// TIA Portal project "pinmachine_vimpr" (V16)

(* hardware
DEVICE "S7-1200 station_1"  S7-1200 Station
   slot 0: "Rack_0"  S7-1200 Rack  Rack  V1.0
   slot 1: "PLC_1"  CPU 1212C DC/DC/DC  6ES7 212-1AE40-0XB0  V4.4
   slot 2: "DI 16x24VDC_1"  6ES7 221-1BH32-0XB0  V2.0
*)

// ===== PLC "PLC_1"  CPU 1212C DC/DC/DC =====

VAR_GLOBAL   // PLC tag table "Default tag table"
   "Cyc1_Top1_Act" AT %I0.0 : Bool;
   "Cyc2_Top1_Act" AT %I0.1 : Bool;
   "Cyc3_Top1_Act" AT %I0.2 : Bool;
   "Cyc4_Top1_Act" AT %I0.3 : Bool;
   "Cyc1_Bot1_Act" AT %I0.4 : Bool;
   "Cyc2_Bot1_Act" AT %I0.5 : Bool;
   "Cyc3_Bot1_Act" AT %I0.6 : Bool;
   "Cyc4_Bot1_Act" AT %I0.7 : Bool;
   "CycHold_Rep" AT %I1.0 : Bool;
   "CycHold_Act" AT %I1.1 : Bool;
   "Cyc1_Top2_Act" AT %I1.2 : Bool;
   "Cyc2_Top2_Act" AT %I1.3 : Bool;
   "Cyc3_Top2_Act" AT %I1.4 : Bool;
   "Cyc4_Top2_Act" AT %I1.5 : Bool;
   "Cyc5_Top2_Act" AT %I1.6 : Bool;
   "Cyc1_Bot2_Act" AT %I1.7 : Bool;
   "Cyc2_Bot2_Act" AT %I2.0 : Bool;
   "Cyc3_Bot2_Act" AT %I2.1 : Bool;
   "Cyc4_Bot2_Act" AT %I2.2 : Bool;
   "Cyc5_Bot2_Act" AT %I2.3 : Bool;
   "Foot_Switch" AT %I2.4 : Bool;
   "4_Part_Detect" AT %I2.5 : Bool;
   "5_Part_Detect" AT %I2.6 : Bool;
   "Safety_Sensor" AT %I2.7 : Bool;
   "QValve4" AT %Q0.0 : Bool;
   "QValve5" AT %Q0.1 : Bool;
   "QHold4" AT %Q0.2 : Bool;
   "QHold5" AT %Q0.3 : Bool;
   "QValveHolder" AT %Q0.4 : Bool;
   "QValveBuzzer" AT %Q0.5 : Bool;
   "MValve4" AT %M0.0 : Bool;
   "MValve5" AT %M0.1 : Bool;
   "MHold4" AT %M0.2 : Bool;
   "MHold5" AT %M0.3 : Bool;
   "x" AT %M0.4 : Bool;
   "MBuzzer" AT %M0.5 : Bool;
   "MBussy" AT %M0.6 : Bool;
   "MDone" AT %M0.7 : Bool;
   "Start" AT %M1.0 : Bool;
   "Auto" AT %M1.1 : Bool;
   "Run" AT %M1.2 : Bool;
   "Timer_Alarm" AT %MD0 : Time;
   "Timer_4Cyl" AT %MD20 : Time;
   "Timer_5Cyl" AT %MD21 : Time;
   "DoneCheckSSBot1" AT %M9.0 : Bool;
   "DoneCheckSSTop1" AT %M9.1 : Bool;
   "DoneCheckSSBot2" AT %M9.2 : Bool;
   "DoneCheckSSTop2" AT %M9.3 : Bool;
   "Alarm" AT %M9.4 : Bool;
   "Cyc1_Top1_Act_Alarm" AT %M9.5 : Bool;
   "Cyc2_Top1_Act_Alarm" AT %M9.6 : Bool;
   "Cyc3_Top1_Act_Alarm" AT %M9.7 : Bool;
   "Cyc4_Top1_Act_Alarm" AT %M10.0 : Bool;
   "Cyc1_Bot1_Act_Alarm" AT %M10.1 : Bool;
   "Cyc2_Bot1_Act_Alarm" AT %M10.2 : Bool;
   "Cyc3_Bot1_Act_Alarm" AT %M10.3 : Bool;
   "Cyc4_Bot1_Act_Alarm" AT %M10.4 : Bool;
   "Cyc1_Bot2_Act_Alarm" AT %M10.5 : Bool;
   "Cyc2_Bot2_Act_Alarm" AT %M10.6 : Bool;
   "Cyc3_Bot2_Act_Alarm" AT %M10.7 : Bool;
   "Cyc4_Bot2_Act_Alarm" AT %M11.0 : Bool;
   "Cyc5_Bot2_Act_Alarm" AT %M11.1 : Bool;
   "Cyc1_Top2_Act_Alarm" AT %M11.2 : Bool;
   "Cyc2_Top2_Act_Alarm" AT %M11.3 : Bool;
   "Cyc3_Top2_Act_Alarm" AT %M11.4 : Bool;
   "Cyc4_Top2_Act_Alarm" AT %M11.5 : Bool;
   "Cyc5_Top2_Act_Alarm" AT %M11.6 : Bool;
   "ResetAlarm" AT %M11.7 : Bool;
   "Step" AT %MW12 : Int;
   "4_Done" AT %M14.0 : Bool;
   "5_Done" AT %M14.1 : Bool;
   "Tag_1" AT %M1000.0 : Bool;
   "Tag_2" AT %M1000.1 : Bool;
   "Tag_3" AT %M1000.3 : Bool;
   "Tag_4" AT %M14.2 : Bool;
   "Tag_5" AT %M14.3 : Bool;
   "Count" AT %MW16 : Int;
   "Tag_6" AT %M1000.4 : Bool;
   "Tag_7" AT %M1000.5 : Bool;
   "Tag_8" AT %M1000.6 : Bool;
   "Tag_9" AT %M1000.7 : Bool;
   "Tag_10" AT %M1001.0 : Bool;
   "Tag_11" AT %M1001.2 : Bool;
   "Tag_12" AT %M1005.1 : Bool;
   "Tag_13" AT %M1005.2 : Bool;
   "Tag_14" AT %M1001.7 : Bool;
   "Tag_15" AT %M1001.6 : Bool;
   "Tag_16" AT %M1007.0 : Bool;
   "Tag_17" AT %M1007.1 : Bool;
END_VAR

DATA_BLOCK "TimerDB"   // DB6
{ S7_Optimized_Access := 'TRUE' }
VERSION : 0.1
   VAR RETAIN
      TimerCyl4_1 : DInt := 1000;
      TimerCyl4_2 : DInt := 1000;
      TimerCyl4_3 : DInt := 1000;
      TimerCyl4_4 : DInt := 1000;
      TimerCyl5_1 : DInt := 1000;
      TimerCyl5_2 : DInt := 1000;
      TimerCyl5_3 : DInt := 1000;
      TimerCyl5_4 : DInt := 1000;
      Timer_Safety : DInt := 5000;
   END_VAR
BEGIN
END_DATA_BLOCK

DATA_BLOCK "AlarmDB"   // DB7
{ S7_Optimized_Access := 'TRUE' }
VERSION : 0.1
   VAR
      Cyc1_Bot1_Act_Alarm : Bool;
      Cyc1_Bot2_Act_Alarm : Bool;
      Cyc1_Bot3_Act_Alarm : Bool;
      Cyc1_Bot4_Act_Alarm : Bool;
      Cyc1_Top1_Act_Alarm : Bool;
      Cyc1_Top2_Act_Alarm : Bool;
      Cyc1_Top3_Act_Alarm : Bool;
      Cyc1_Top4_Act_Alarm : Bool;
      Cyc2_Bot1_Act_Alarm : Bool;
      Cyc2_Bot2_Act_Alarm : Bool;
      Cyc2_Bot3_Act_Alarm : Bool;
      Cyc2_Bot4_Act_Alarm : Bool;
      Cyc2_Bot5_Act_Alarm : Bool;
      Cyc2_Top1_Act_Alarm : Bool;
      Cyc2_Top2_Act_Alarm : Bool;
      Cyc2_Top3_Act_Alarm : Bool;
      Cyc2_Top4_Act_Alarm : Bool;
      Cyc2_Top5_Act_Alarm : Bool;
      Sensor_Detect_4 : Bool;
      Sensor_Detect_5 : Bool;
      Sensor_Safety : Bool;
   END_VAR
BEGIN
END_DATA_BLOCK

// folder: System blocks/Program resources

DATA_BLOCK "TimerDone45"   // DB1
{ S7_Optimized_Access := 'TRUE' }
AUTHOR : Simatic
FAMILY : IEC
NAME : IEC_TMR
VERSION : 1.0
// stored: InstanceOfName IEC_TIMER
"IEC_TIMER"
BEGIN
END_DATA_BLOCK

DATA_BLOCK "TimerError"   // DB5
{ S7_Optimized_Access := 'TRUE' }
AUTHOR : Simatic
FAMILY : IEC
NAME : IEC_TMR
VERSION : 1.0
// stored: InstanceOfName IEC_TIMER
"IEC_TIMER"
BEGIN
END_DATA_BLOCK

DATA_BLOCK "TimerResetAlarm"   // DB16
{ S7_Optimized_Access := 'TRUE' }
AUTHOR : Simatic
FAMILY : IEC
NAME : IEC_TMR
VERSION : 1.0
// stored: InstanceOfName IEC_TIMER
"IEC_TIMER"
BEGIN
END_DATA_BLOCK

DATA_BLOCK "TimerResetStep"   // DB17
{ S7_Optimized_Access := 'TRUE' }
AUTHOR : Simatic
FAMILY : IEC
NAME : IEC_TMR
VERSION : 1.0
// stored: InstanceOfName IEC_TIMER
"IEC_TIMER"
BEGIN
END_DATA_BLOCK

// folder: (top level)

ORGANIZATION_BLOCK "Main"   // OB1, LAD, ProgramCycle
TITLE = "Main Program Sweep (Cycle)"
{ S7_Optimized_Access := 'TRUE' }
VERSION : 0.1
   VAR_INPUT
      Initial_Call : Bool;   // Initial call of this OB
      Remanence : Bool;   // =True, if remanent data are available
   END_VAR
   VAR_TEMP   // added for the SCL form of the ladder/FBD networks
      _w1 : Bool;
      _w2 : Bool;
      _w3 : Bool;
      _w4 : Bool;
      _w5 : Bool;
   END_VAR
BEGIN

REGION Network 1: Cycle
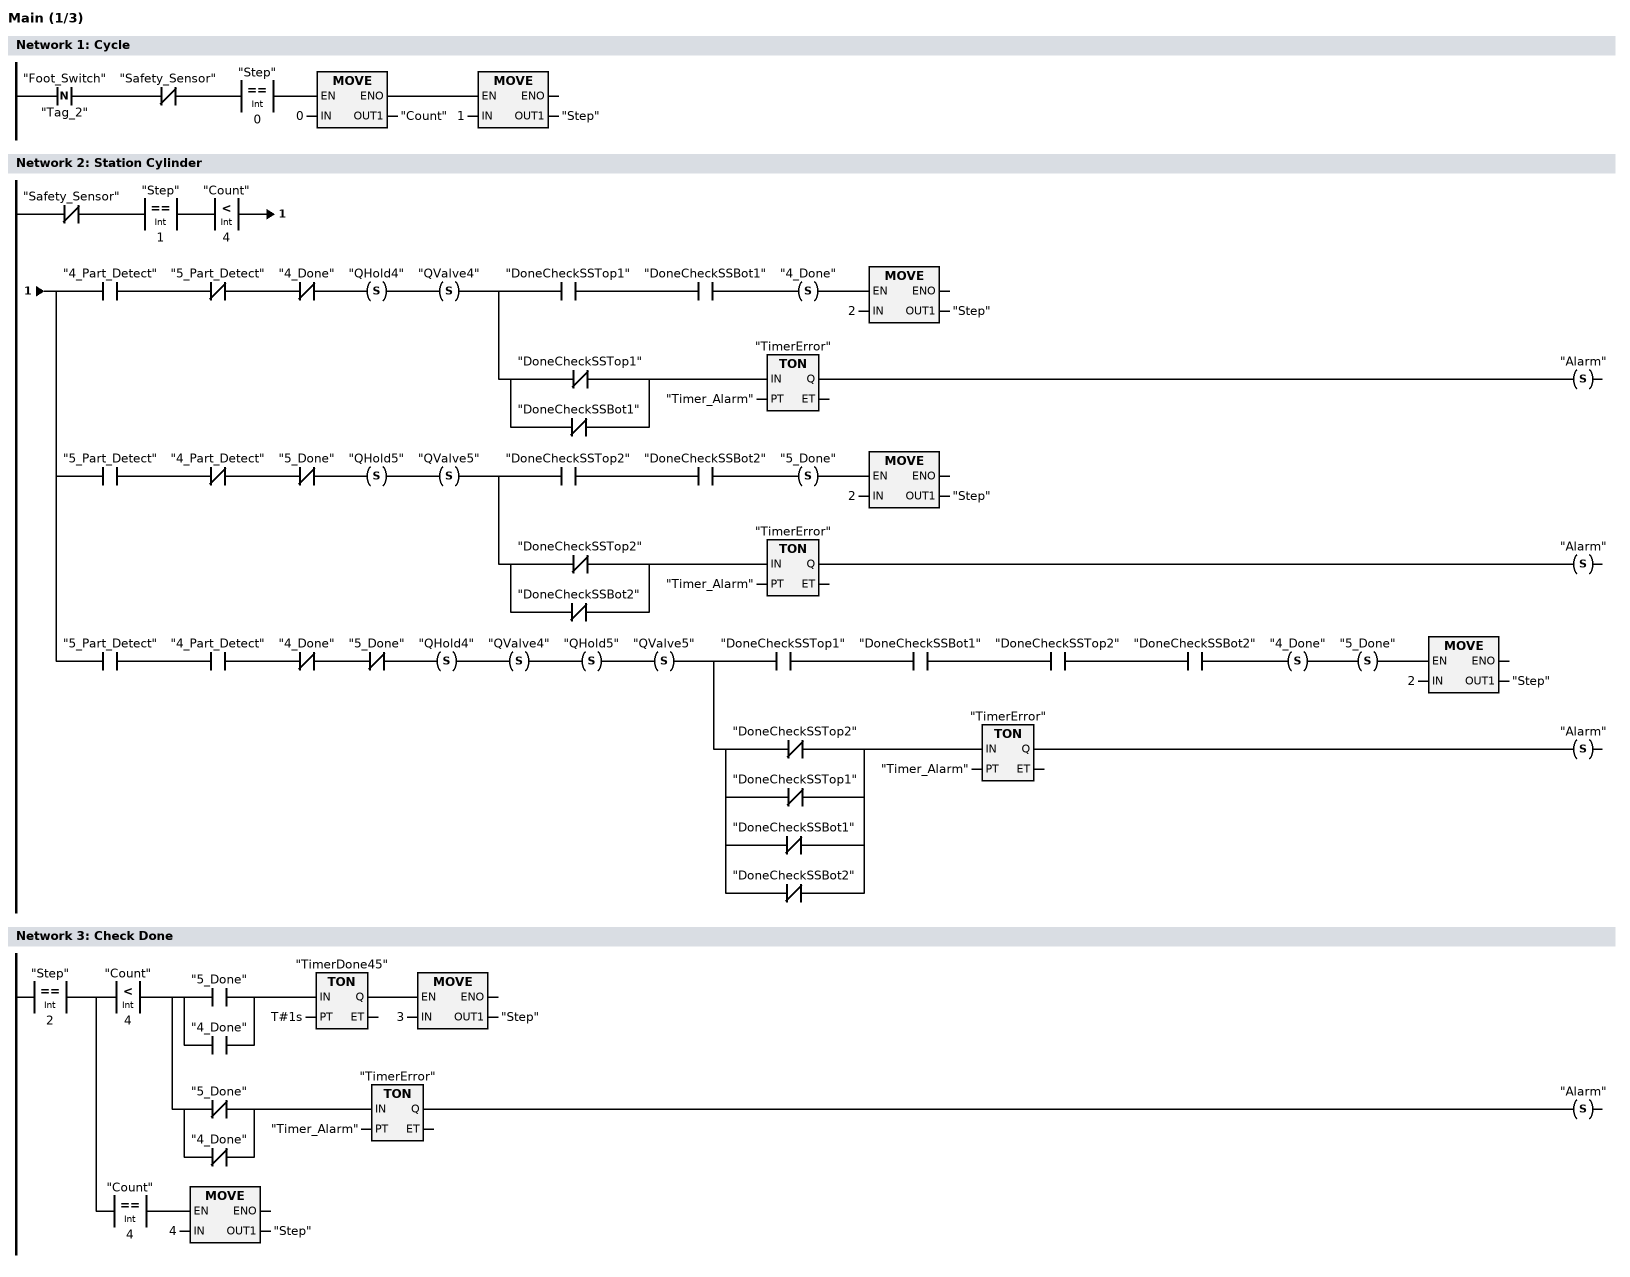
   RUNG wire#powerrail
      N_Contact(operand := "Foot_Switch", bit := "Tag_2")
      I_Contact( "Safety_Sensor" )
      { S7_Templates := "SrcType := Int" } EQ_Contact(in1 := "Step", in2 := 0)
      Move(in := 0, out1 => "Count")
      Move(in := 1, out1 => "Step")
   END_RUNG
   // the same network as SCL:
   #_w1 := NOT "Foot_Switch" AND "Tag_2";   // falling edge of "Foot_Switch"
   "Tag_2" := "Foot_Switch";
   IF #_w1 AND NOT "Safety_Sensor" AND ("Step" = 0) THEN
       "Count" := 0;
       "Step" := 1;
   END_IF;
END_REGION

REGION Network 2: Station Cylinder
   #_w1 := NOT "Safety_Sensor" AND ("Step" = 1) AND ("Count" < 4);
   #_w2 := #_w1 AND "4_Part_Detect" AND NOT "5_Part_Detect" AND NOT "4_Done";
   IF #_w2 THEN
       "QHold4" := TRUE;
       "QValve4" := TRUE;
   END_IF;
   IF #_w2 AND "DoneCheckSSTop1" AND "DoneCheckSSBot1" THEN
       "4_Done" := TRUE;
       "Step" := 2;
   END_IF;
   "TimerError".TON(IN := #_w2 AND (NOT "DoneCheckSSTop1" OR NOT "DoneCheckSSBot1"), PT := "Timer_Alarm");
   IF "TimerError".Q THEN "Alarm" := TRUE; END_IF;
   #_w3 := #_w1 AND "5_Part_Detect" AND NOT "4_Part_Detect" AND NOT "5_Done";
   IF #_w3 THEN
       "QHold5" := TRUE;
       "QValve5" := TRUE;
   END_IF;
   IF #_w3 AND "DoneCheckSSTop2" AND "DoneCheckSSBot2" THEN
       "5_Done" := TRUE;
       "Step" := 2;
   END_IF;
   "TimerError".TON(IN := #_w3 AND (NOT "DoneCheckSSTop2" OR NOT "DoneCheckSSBot2"), PT := "Timer_Alarm");
   IF "TimerError".Q THEN "Alarm" := TRUE; END_IF;
   #_w4 := #_w1 AND "5_Part_Detect" AND "4_Part_Detect" AND NOT "4_Done" AND NOT "5_Done";
   IF #_w4 THEN
       "QHold4" := TRUE;
       "QValve4" := TRUE;
       "QHold5" := TRUE;
       "QValve5" := TRUE;
   END_IF;
   IF #_w4 AND "DoneCheckSSTop1" AND "DoneCheckSSBot1" AND "DoneCheckSSTop2" AND "DoneCheckSSBot2" THEN
       "4_Done" := TRUE;
       "5_Done" := TRUE;
       "Step" := 2;
   END_IF;
   "TimerError".TON(IN := #_w4 AND (NOT "DoneCheckSSTop2" OR NOT "DoneCheckSSTop1" OR NOT "DoneCheckSSBot1" OR NOT "DoneCheckSSBot2"),
                    PT := "Timer_Alarm");
   IF "TimerError".Q THEN "Alarm" := TRUE; END_IF;
END_REGION

REGION Network 3: Check Done
   #_w1 := "Step" = 2;
   #_w2 := #_w1 AND ("Count" < 4);
   "TimerDone45".TON(IN := #_w2 AND ("5_Done" OR "4_Done"), PT := T#1s);
   IF "TimerDone45".Q THEN "Step" := 3; END_IF;
   "TimerError".TON(IN := #_w2 AND (NOT "5_Done" OR NOT "4_Done"), PT := "Timer_Alarm");
   IF "TimerError".Q THEN "Alarm" := TRUE; END_IF;
   IF #_w1 AND ("Count" = 4) THEN "Step" := 4; END_IF;
END_REGION

REGION Network 4: Step Reset Valve
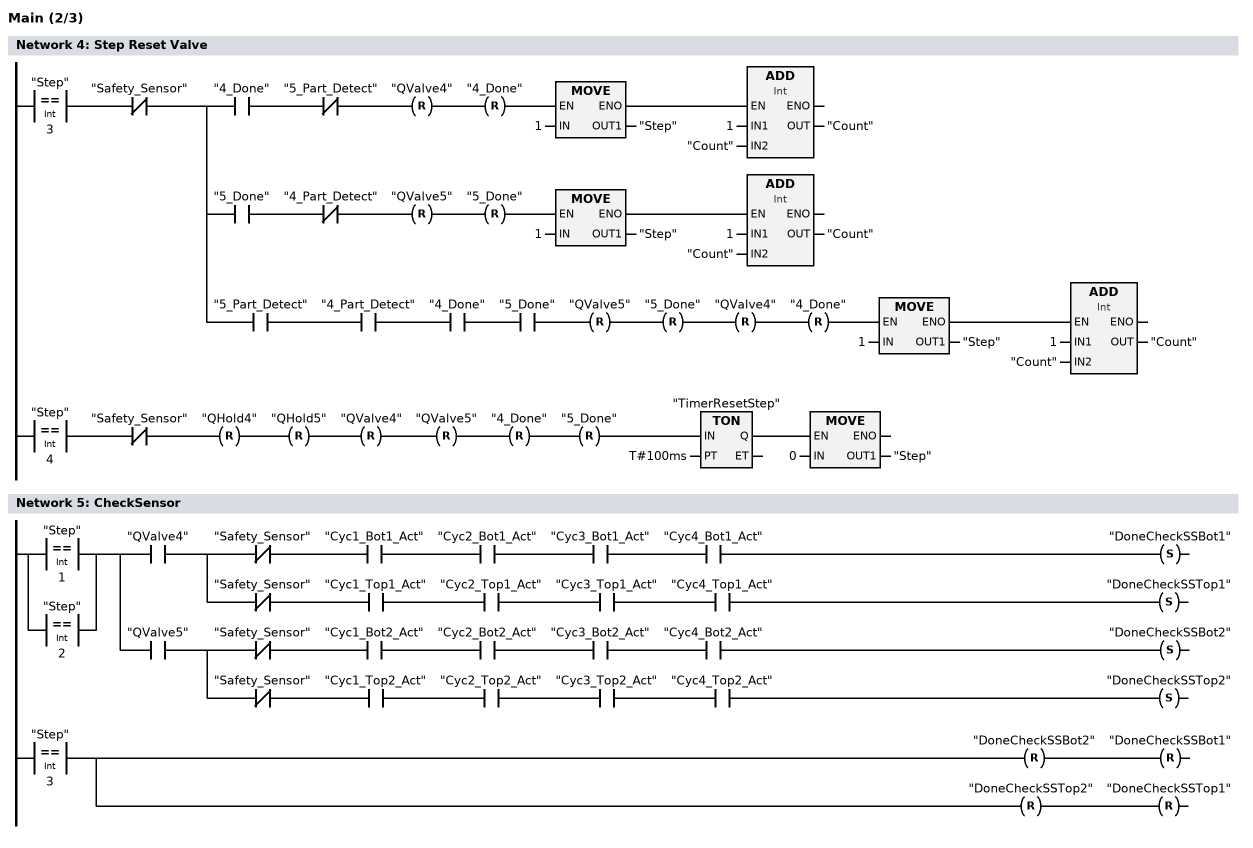
   #_w1 := ("Step" = 3) AND NOT "Safety_Sensor";
   IF #_w1 AND "4_Done" AND NOT "5_Part_Detect" THEN "QValve4" := FALSE; END_IF;
   #_w2 := #_w1 AND "4_Done" AND NOT "5_Part_Detect";
   IF #_w2 THEN
       "4_Done" := FALSE;
       "Step" := 1;
       "Count" := 1 + "Count";
   END_IF;
   IF #_w1 AND "5_Done" AND NOT "4_Part_Detect" THEN "QValve5" := FALSE; END_IF;
   #_w3 := #_w1 AND "5_Done" AND NOT "4_Part_Detect";
   IF #_w3 THEN
       "5_Done" := FALSE;
       "Step" := 1;
       "Count" := 1 + "Count";
   END_IF;
   IF #_w1 AND "5_Part_Detect" AND "4_Part_Detect" AND "4_Done" AND "5_Done" THEN "QValve5" := FALSE; END_IF;
   #_w4 := #_w1 AND "5_Part_Detect" AND "4_Part_Detect" AND "4_Done" AND "5_Done";
   IF #_w4 THEN
       "5_Done" := FALSE;
       "QValve4" := FALSE;
       "4_Done" := FALSE;
       "Step" := 1;
       "Count" := 1 + "Count";
   END_IF;
   #_w5 := ("Step" = 4) AND NOT "Safety_Sensor";
   IF #_w5 THEN
       "QHold4" := FALSE;
       "QHold5" := FALSE;
       "QValve4" := FALSE;
       "QValve5" := FALSE;
       "4_Done" := FALSE;
       "5_Done" := FALSE;
   END_IF;
   "TimerResetStep".TON(IN := #_w5, PT := T#100ms);
   IF "TimerResetStep".Q THEN "Step" := 0; END_IF;
END_REGION

REGION Network 5: CheckSensor
   RUNG wire#powerrail
      { S7_Templates := "SrcType := Int" } EQ_Contact(in1 := "Step", in2 := 1)
      wire#w1
      Contact( "QValve4" )
      wire#w2
      I_Contact( "Safety_Sensor" )
      Contact( "Cyc1_Bot1_Act" )
      Contact( "Cyc2_Bot1_Act" )
      Contact( "Cyc3_Bot1_Act" )
      Contact( "Cyc4_Bot1_Act" )
      S_Coil( "DoneCheckSSBot1" )
   END_RUNG
   RUNG wire#powerrail
      { S7_Templates := "SrcType := Int" } EQ_Contact(in1 := "Step", in2 := 2)
   END_RUNG wire#w1
   RUNG wire#w2
      I_Contact( "Safety_Sensor" )
      Contact( "Cyc1_Top1_Act" )
      Contact( "Cyc2_Top1_Act" )
      Contact( "Cyc3_Top1_Act" )
      Contact( "Cyc4_Top1_Act" )
      S_Coil( "DoneCheckSSTop1" )
   END_RUNG
   RUNG wire#w1
      Contact( "QValve5" )
      wire#w3
      I_Contact( "Safety_Sensor" )
      Contact( "Cyc1_Bot2_Act" )
      Contact( "Cyc2_Bot2_Act" )
      Contact( "Cyc3_Bot2_Act" )
      Contact( "Cyc4_Bot2_Act" )
      S_Coil( "DoneCheckSSBot2" )
   END_RUNG
   RUNG wire#w3
      I_Contact( "Safety_Sensor" )
      Contact( "Cyc1_Top2_Act" )
      Contact( "Cyc2_Top2_Act" )
      Contact( "Cyc3_Top2_Act" )
      Contact( "Cyc4_Top2_Act" )
      S_Coil( "DoneCheckSSTop2" )
   END_RUNG
   RUNG wire#powerrail
      { S7_Templates := "SrcType := Int" } EQ_Contact(in1 := "Step", in2 := 3)
      wire#w4
      R_Coil( "DoneCheckSSBot2" )
      R_Coil( "DoneCheckSSBot1" )
   END_RUNG
   RUNG wire#w4
      R_Coil( "DoneCheckSSTop2" )
      R_Coil( "DoneCheckSSTop1" )
   END_RUNG
   // the same network as SCL:
   #_w1 := ("Step" = 1) OR ("Step" = 2);
   #_w2 := #_w1 AND "QValve4";
   IF #_w2 AND NOT "Safety_Sensor" AND "Cyc1_Bot1_Act" AND "Cyc2_Bot1_Act" AND "Cyc3_Bot1_Act" AND "Cyc4_Bot1_Act" THEN
       "DoneCheckSSBot1" := TRUE;
   END_IF;
   IF #_w2 AND NOT "Safety_Sensor" AND "Cyc1_Top1_Act" AND "Cyc2_Top1_Act" AND "Cyc3_Top1_Act" AND "Cyc4_Top1_Act" THEN
       "DoneCheckSSTop1" := TRUE;
   END_IF;
   #_w3 := #_w1 AND "QValve5";
   IF #_w3 AND NOT "Safety_Sensor" AND "Cyc1_Bot2_Act" AND "Cyc2_Bot2_Act" AND "Cyc3_Bot2_Act" AND "Cyc4_Bot2_Act" THEN
       "DoneCheckSSBot2" := TRUE;
   END_IF;
   IF #_w3 AND NOT "Safety_Sensor" AND "Cyc1_Top2_Act" AND "Cyc2_Top2_Act" AND "Cyc3_Top2_Act" AND "Cyc4_Top2_Act" THEN
       "DoneCheckSSTop2" := TRUE;
   END_IF;
   IF "Step" = 3 THEN
       "DoneCheckSSBot2" := FALSE;
       "DoneCheckSSBot1" := FALSE;
       "DoneCheckSSTop2" := FALSE;
       "DoneCheckSSTop1" := FALSE;
   END_IF;
END_REGION

REGION Network 6: Alarm
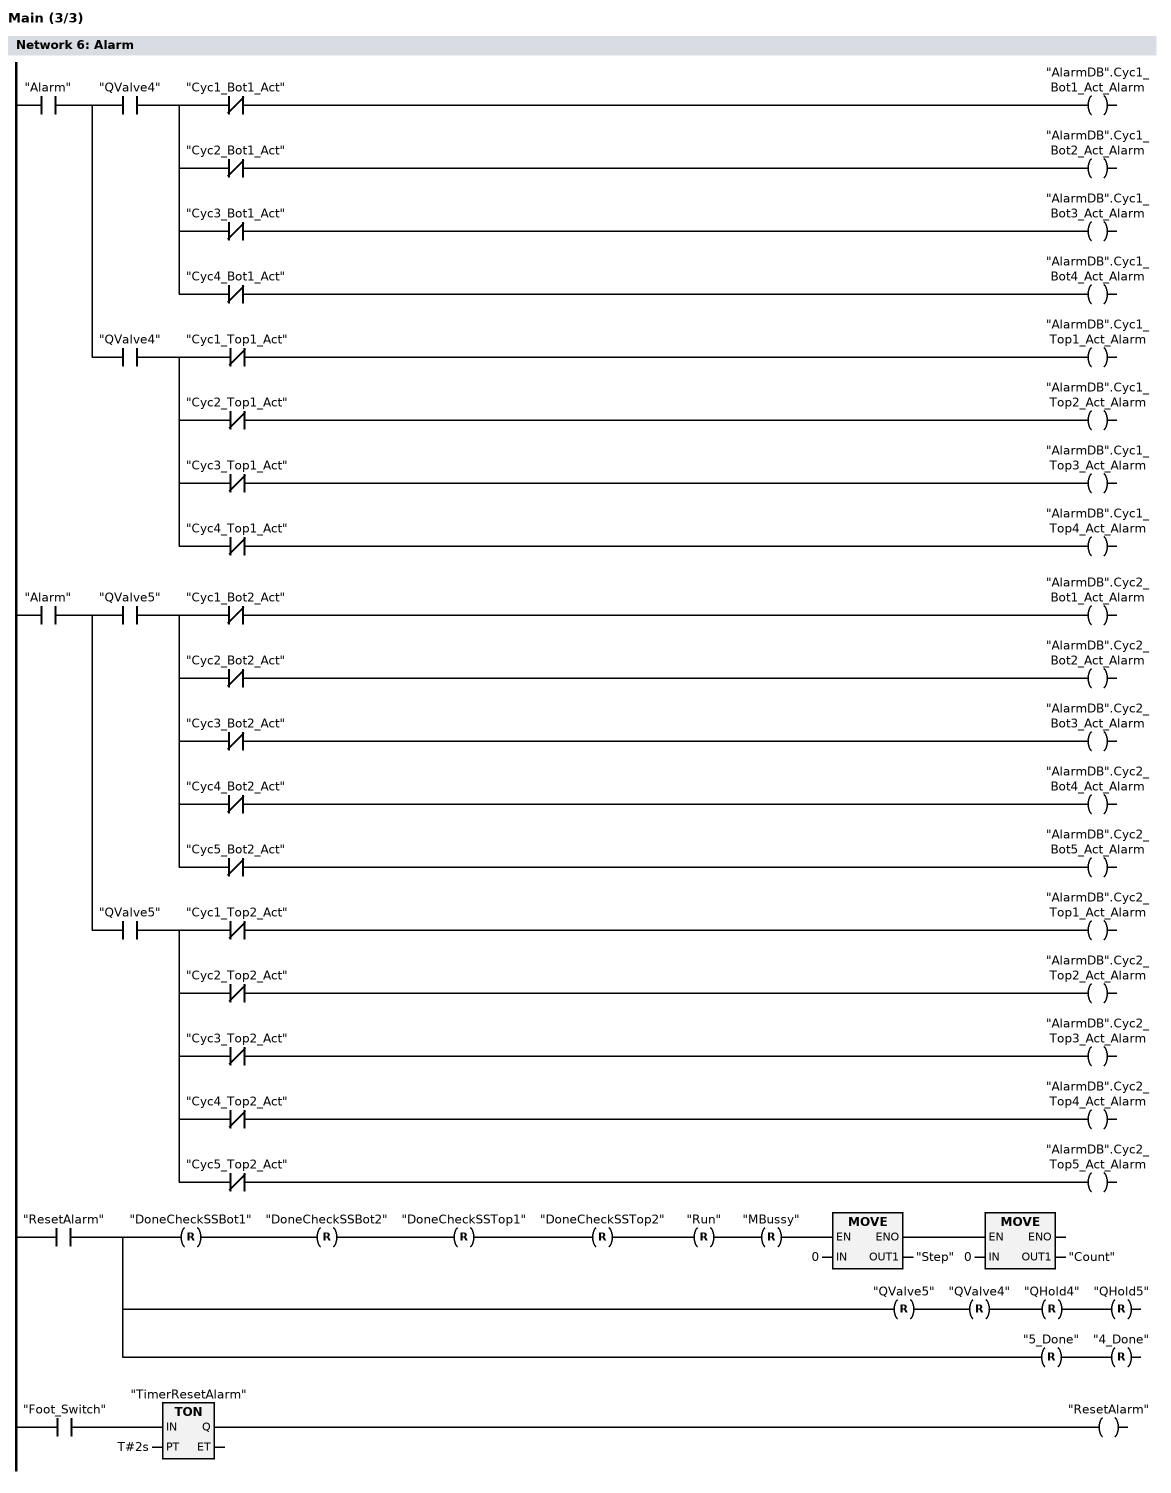
   #_w1 := "Alarm" AND "QValve4";
   "AlarmDB".Cyc1_Bot1_Act_Alarm := #_w1 AND NOT "Cyc1_Bot1_Act";
   "AlarmDB".Cyc1_Bot2_Act_Alarm := #_w1 AND NOT "Cyc2_Bot1_Act";
   "AlarmDB".Cyc1_Bot3_Act_Alarm := #_w1 AND NOT "Cyc3_Bot1_Act";
   "AlarmDB".Cyc1_Bot4_Act_Alarm := #_w1 AND NOT "Cyc4_Bot1_Act";
   #_w2 := "Alarm" AND "QValve4";
   "AlarmDB".Cyc1_Top1_Act_Alarm := #_w2 AND NOT "Cyc1_Top1_Act";
   "AlarmDB".Cyc1_Top2_Act_Alarm := #_w2 AND NOT "Cyc2_Top1_Act";
   "AlarmDB".Cyc1_Top3_Act_Alarm := #_w2 AND NOT "Cyc3_Top1_Act";
   "AlarmDB".Cyc1_Top4_Act_Alarm := #_w2 AND NOT "Cyc4_Top1_Act";
   #_w3 := "Alarm" AND "QValve5";
   "AlarmDB".Cyc2_Bot1_Act_Alarm := #_w3 AND NOT "Cyc1_Bot2_Act";
   "AlarmDB".Cyc2_Bot2_Act_Alarm := #_w3 AND NOT "Cyc2_Bot2_Act";
   "AlarmDB".Cyc2_Bot3_Act_Alarm := #_w3 AND NOT "Cyc3_Bot2_Act";
   "AlarmDB".Cyc2_Bot4_Act_Alarm := #_w3 AND NOT "Cyc4_Bot2_Act";
   "AlarmDB".Cyc2_Bot5_Act_Alarm := #_w3 AND NOT "Cyc5_Bot2_Act";
   #_w4 := "Alarm" AND "QValve5";
   "AlarmDB".Cyc2_Top1_Act_Alarm := #_w4 AND NOT "Cyc1_Top2_Act";
   "AlarmDB".Cyc2_Top2_Act_Alarm := #_w4 AND NOT "Cyc2_Top2_Act";
   "AlarmDB".Cyc2_Top3_Act_Alarm := #_w4 AND NOT "Cyc3_Top2_Act";
   "AlarmDB".Cyc2_Top4_Act_Alarm := #_w4 AND NOT "Cyc4_Top2_Act";
   "AlarmDB".Cyc2_Top5_Act_Alarm := #_w4 AND NOT "Cyc5_Top2_Act";
   IF "ResetAlarm" THEN
       "DoneCheckSSBot1" := FALSE;
       "DoneCheckSSBot2" := FALSE;
       "DoneCheckSSTop1" := FALSE;
       "DoneCheckSSTop2" := FALSE;
       "Run" := FALSE;
       "MBussy" := FALSE;
       "Step" := 0;
       "Count" := 0;
       "QValve5" := FALSE;
       "QValve4" := FALSE;
       "QHold4" := FALSE;
       "QHold5" := FALSE;
       "5_Done" := FALSE;
       "4_Done" := FALSE;
   END_IF;
   "TimerResetAlarm".TON(IN := "Foot_Switch", PT := T#2s);
   "ResetAlarm" := "TimerResetAlarm".Q;
END_REGION

REGION Network 7 (SCL): Timer Parameter
   CASE "Count" OF
       1:
           "Timer_4Cyl" := "TimerDB".TimerCyl4_1;
           "Timer_5Cyl" := "TimerDB".TimerCyl5_1;
       2:
           "Timer_4Cyl" := "TimerDB".TimerCyl4_2;
           "Timer_5Cyl" := "TimerDB".TimerCyl5_2;
       3:
           "Timer_4Cyl" := "TimerDB"."TimerCyl4_3";
           "Timer_5Cyl" := "TimerDB".TimerCyl5_3;
       4:
           "Timer_4Cyl" := "TimerDB"."TimerCyl4_4";
           "Timer_5Cyl" := "TimerDB".TimerCyl5_4;
   END_CASE;
END_REGION
END_ORGANIZATION_BLOCK